Universal Robots PolyScope program: test serial 2.urp

Program test serial 2 (installation=default directory=/programs createdIn=5.14.5 lastSavedIn=5.14.5 robotSerialNumber=20236801216)
Calibrated DH parameters: a=[-0.000021, -0.748897, -0.28186, -0.00004, -0.000055, 0]; d=[0.236225, -424.082933, -1564.66872, 1988.95162, 0.159094, 0.153873]; alpha=[1.570844, 0.001002, 0.000337, 1.571488, -1.569996, 0]; deltaTheta=[0, -0.516316, 5.626292, 1.173211, 0.000001, 0]
InitVariablesNode
Robot Program (runOnlyOnce=false)
  SuppressedNode
    URCap WireTank Serial (WireTank Serial, WireTank, LLC) dataModel(Command=[252,72,49], byte_array=true, NODE_TITLE=Serial Bridge uH1, QUERY=false, OUTPUT_ENTRY=Static, Variable(key=OUTPUT_VARIABLE, variable(name=HwResp)))
  URCap WireTank Serial (WireTank Serial, WireTank, LLC) dataModel(byte_array=true, NODE_TITLE=Serial Bridge uR1, Command=[252,82,49], OUTPUT_ENTRY=Static, QUERY=true, Variable(key=OUTPUT_VARIABLE, variable=HwResp))
  Set DigitalOutput pin=digital_out[0]; digitalValue=1
  Script: popup(HwResp)
  SuppressedNode
    Wait Sleep waitTime=5
  Popup Message (haltProgram=false message=on inputType=Text)
  Set DigitalOutput pin=digital_out[0]; digitalValue=0
  URCap WireTank Serial (WireTank Serial, WireTank, LLC) dataModel(NODE_TITLE=Serial Bridge uR0, Command=[252,82,48], byte_array=true, OUTPUT_ENTRY=Static, QUERY=true, Variable(key=OUTPUT_VARIABLE, variable=HwResp))
  Script: popup(HwResp)
  Popup Message (haltProgram=false message=off inputType=Text)
